SYSTEM TestSP
  (* Version 1.0, 2024-01-14, ADMIN *)
  APPLICATION TestSPApp
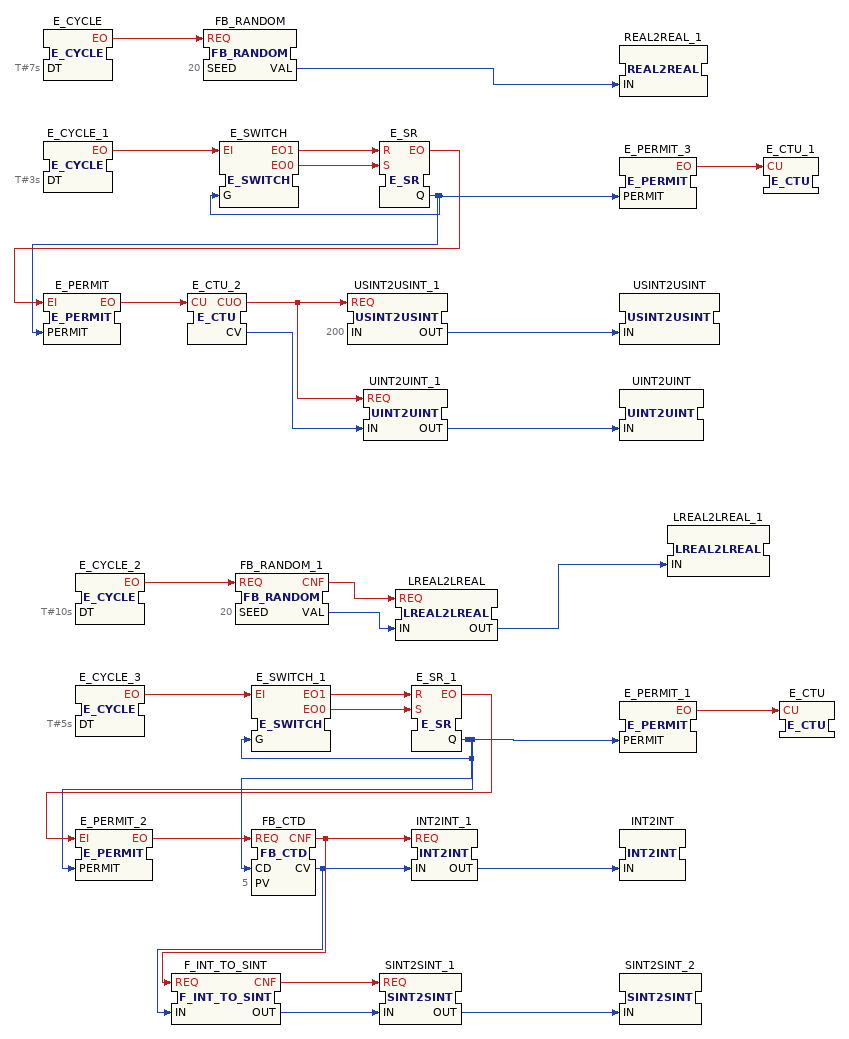
    FBS
      E_CYCLE : E_CYCLE(DT := T#7s);
      FB_RANDOM : FB_RANDOM(SEED := 20);
      E_CYCLE_1 : E_CYCLE(DT := T#3s);
      E_SWITCH : E_SWITCH;
      E_SR : E_SR;
      E_PERMIT : E_PERMIT;
      E_PERMIT_1 : E_PERMIT;
      E_CTU : E_CTU;
      E_CYCLE_2 : E_CYCLE(DT := T#10s);
      FB_RANDOM_1 : FB_RANDOM(SEED := 20);
      E_CYCLE_3 : E_CYCLE(DT := T#5s);
      E_SWITCH_1 : E_SWITCH;
      E_SR_1 : E_SR;
      E_PERMIT_2 : E_PERMIT;
      REAL2REAL_1 : REAL2REAL;
      E_PERMIT_3 : E_PERMIT;
      E_CTU_1 : E_CTU;
      UINT2UINT : UINT2UINT;
      INT2INT : INT2INT;
      SINT2SINT_1 : SINT2SINT;
      USINT2USINT : USINT2USINT;
      E_CTU_2 : E_CTU;
      UINT2UINT_1 : UINT2UINT;
      SINT2SINT_2 : SINT2SINT;
      INT2INT_1 : INT2INT;
      USINT2USINT_1 : USINT2USINT(IN := 200);
      LREAL2LREAL : LREAL2LREAL;
      LREAL2LREAL_1 : LREAL2LREAL;
      FB_CTD : FB_CTD(PV := 5);
      F_INT_TO_SINT : F_INT_TO_SINT;
    END_FBS
    EVENT_CONNECTIONS
      E_CYCLE.EO TO FB_RANDOM.REQ;
      E_SWITCH.EO1 TO E_SR.R;
      E_SWITCH.EO0 TO E_SR.S;
      E_SR.EO TO E_PERMIT.EI;
      E_CYCLE_1.EO TO E_SWITCH.EI;
      E_PERMIT_1.EO TO E_CTU.CU;
      E_PERMIT_3.EO TO E_CTU_1.CU;
      E_SR_1.EO TO E_PERMIT_2.EI;
      E_CYCLE_2.EO TO FB_RANDOM_1.REQ;
      E_SWITCH_1.EO1 TO E_SR_1.R;
      E_CYCLE_3.EO TO E_SWITCH_1.EI;
      E_SWITCH_1.EO0 TO E_SR_1.S;
      E_PERMIT.EO TO E_CTU_2.CU;
      E_CTU_2.CUO TO UINT2UINT_1.REQ;
      E_CTU_2.CUO TO USINT2USINT_1.REQ;
      FB_RANDOM_1.CNF TO LREAL2LREAL.REQ;
      E_PERMIT_2.EO TO FB_CTD.REQ;
      FB_CTD.CNF TO INT2INT_1.REQ;
      F_INT_TO_SINT.CNF TO SINT2SINT_1.REQ;
      FB_CTD.CNF TO F_INT_TO_SINT.REQ;
    END_CONNECTIONS
    DATA_CONNECTIONS
      E_SR.Q TO E_SWITCH.G;
      E_SR.Q TO E_PERMIT.PERMIT;
      E_SR_1.Q TO E_SWITCH_1.G;
      E_SR_1.Q TO E_PERMIT_2.PERMIT;
      E_SR.Q TO E_PERMIT_3.PERMIT;
      E_SR_1.Q TO E_PERMIT_1.PERMIT;
      FB_RANDOM.VAL TO REAL2REAL_1.IN;
      E_CTU_2.CV TO UINT2UINT_1.IN;
      INT2INT_1.OUT TO INT2INT.IN;
      SINT2SINT_1.OUT TO SINT2SINT_2.IN;
      USINT2USINT_1.OUT TO USINT2USINT.IN;
      UINT2UINT_1.OUT TO UINT2UINT.IN;
      FB_RANDOM_1.VAL TO LREAL2LREAL.IN;
      LREAL2LREAL.OUT TO LREAL2LREAL_1.IN;
      FB_CTD.CV TO INT2INT_1.IN;
      F_INT_TO_SINT.OUT TO SINT2SINT_1.IN;
      FB_CTD.CV TO F_INT_TO_SINT.IN;
      E_SR_1.Q TO FB_CTD.CD;
    END_CONNECTIONS
  END_APPLICATION
  DEVICE BeagleBoneBlack : BeagleBoneBlack(MGR_ID := "localhost:61500")
    {SET_ATTRIBUTE(Profile, HOLOBLOC)} (* device profile *)
    RESOURCE EMB_RES : EMB_RES
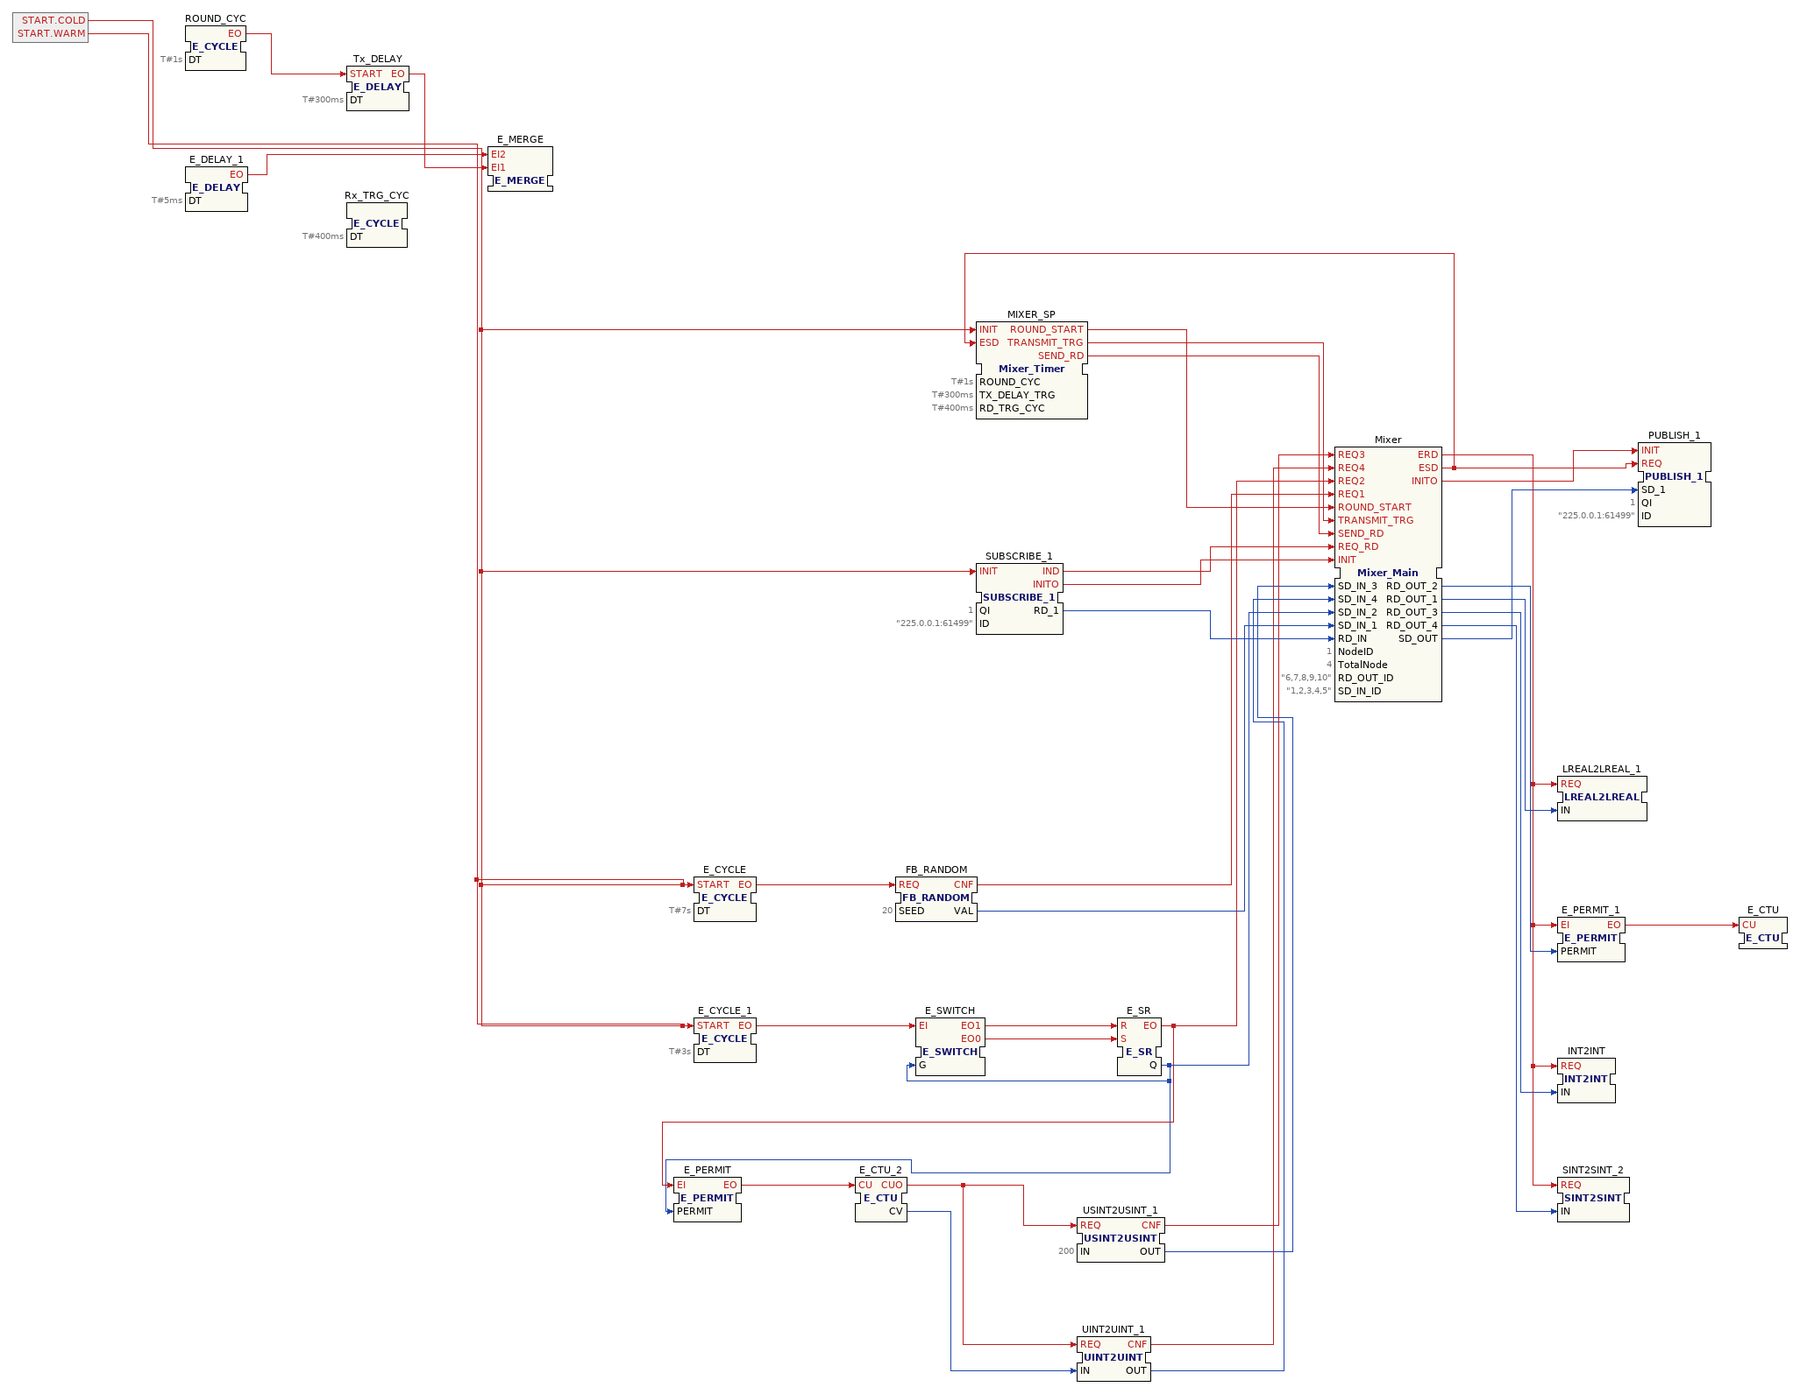
      FBS
        Mixer : Mixer_Main(NodeID := 1, TotalNode := 4, RD_OUT_ID := "6,7,8,9,10", SD_IN_ID := "1,2,3,4,5");
        Rx_TRG_CYC : E_CYCLE(DT := T#400ms);
        PUBLISH_1 : PUBLISH_1(QI := 1, ID := "225.0.0.1:61499");
        E_DELAY_1 : E_DELAY(DT := T#5ms);
        SUBSCRIBE_1 : SUBSCRIBE_1(QI := 1, ID := "225.0.0.1:61499");
        E_MERGE : E_MERGE;
        Tx_DELAY : E_DELAY(DT := T#300ms);
        ROUND_CYC : E_CYCLE(DT := T#1s);
        USINT2USINT_1 : USINT2USINT(IN := 200);
        UINT2UINT_1 : UINT2UINT;
        E_CTU_2 : E_CTU;
        E_CTU : E_CTU;
        E_PERMIT_1 : E_PERMIT;
        E_PERMIT : E_PERMIT;
        E_SR : E_SR;
        E_SWITCH : E_SWITCH;
        E_CYCLE_1 : E_CYCLE(DT := T#3s);
        FB_RANDOM : FB_RANDOM(SEED := 20);
        E_CYCLE : E_CYCLE(DT := T#7s);
        LREAL2LREAL_1 : LREAL2LREAL;
        INT2INT : INT2INT;
        SINT2SINT_2 : SINT2SINT;
        MIXER_SP : Mixer_Timer(ROUND_CYC := T#1s, TX_DELAY_TRG := T#300ms, RD_TRG_CYC := T#400ms);
      END_FBS
      EVENT_CONNECTIONS
        ROUND_CYC.EO TO Tx_DELAY.START;
        E_DELAY_1.EO TO E_MERGE.EI2;
        Tx_DELAY.EO TO E_MERGE.EI1;
        USINT2USINT_1.CNF TO Mixer.REQ3;
        UINT2UINT_1.CNF TO Mixer.REQ4;
        E_CTU_2.CUO TO UINT2UINT_1.REQ;
        E_CTU_2.CUO TO USINT2USINT_1.REQ;
        E_PERMIT_1.EO TO E_CTU.CU;
        Mixer.ERD TO E_PERMIT_1.EI;
        E_PERMIT.EO TO E_CTU_2.CU;
        E_SR.EO TO E_PERMIT.EI;
        E_SR.EO TO Mixer.REQ2;
        E_SWITCH.EO1 TO E_SR.R;
        E_SWITCH.EO0 TO E_SR.S;
        E_CYCLE_1.EO TO E_SWITCH.EI;
        START.COLD TO E_CYCLE_1.START;
        START.WARM TO E_CYCLE_1.START;
        FB_RANDOM.CNF TO Mixer.REQ1;
        E_CYCLE.EO TO FB_RANDOM.REQ;
        START.COLD TO E_CYCLE.START;
        START.WARM TO E_CYCLE.START;
        Mixer.ERD TO LREAL2LREAL_1.REQ;
        Mixer.ERD TO INT2INT.REQ;
        Mixer.ERD TO SINT2SINT_2.REQ;
        START.COLD TO MIXER_SP.INIT;
        Mixer.ESD TO MIXER_SP.ESD;
        MIXER_SP.ROUND_START TO Mixer.ROUND_START;
        MIXER_SP.TRANSMIT_TRG TO Mixer.TRANSMIT_TRG;
        MIXER_SP.SEND_RD TO Mixer.SEND_RD;
        SUBSCRIBE_1.IND TO Mixer.REQ_RD;
        Mixer.INITO TO PUBLISH_1.INIT;
        Mixer.ESD TO PUBLISH_1.REQ;
        SUBSCRIBE_1.INITO TO Mixer.INIT;
        START.COLD TO SUBSCRIBE_1.INIT;
      END_CONNECTIONS
      DATA_CONNECTIONS
        USINT2USINT_1.OUT TO Mixer.SD_IN_3;
        UINT2UINT_1.OUT TO Mixer.SD_IN_4;
        E_CTU_2.CV TO UINT2UINT_1.IN;
        E_SR.Q TO E_PERMIT.PERMIT;
        E_SR.Q TO Mixer.SD_IN_2;
        E_SR.Q TO E_SWITCH.G;
        FB_RANDOM.VAL TO Mixer.SD_IN_1;
        Mixer.RD_OUT_2 TO E_PERMIT_1.PERMIT;
        Mixer.RD_OUT_1 TO LREAL2LREAL_1.IN;
        Mixer.RD_OUT_3 TO INT2INT.IN;
        Mixer.RD_OUT_4 TO SINT2SINT_2.IN;
        SUBSCRIBE_1.RD_1 TO Mixer.RD_IN;
        Mixer.SD_OUT TO PUBLISH_1.SD_1;
      END_CONNECTIONS
    END_RESOURCE
  END_DEVICE
  DEVICE BeagleBoneBlack_1 : BeagleBoneBlack(MGR_ID := "localhost:61501")
    {SET_ATTRIBUTE(Profile, HOLOBLOC)} (* device profile *)
    RESOURCE EMB_RES : EMB_RES
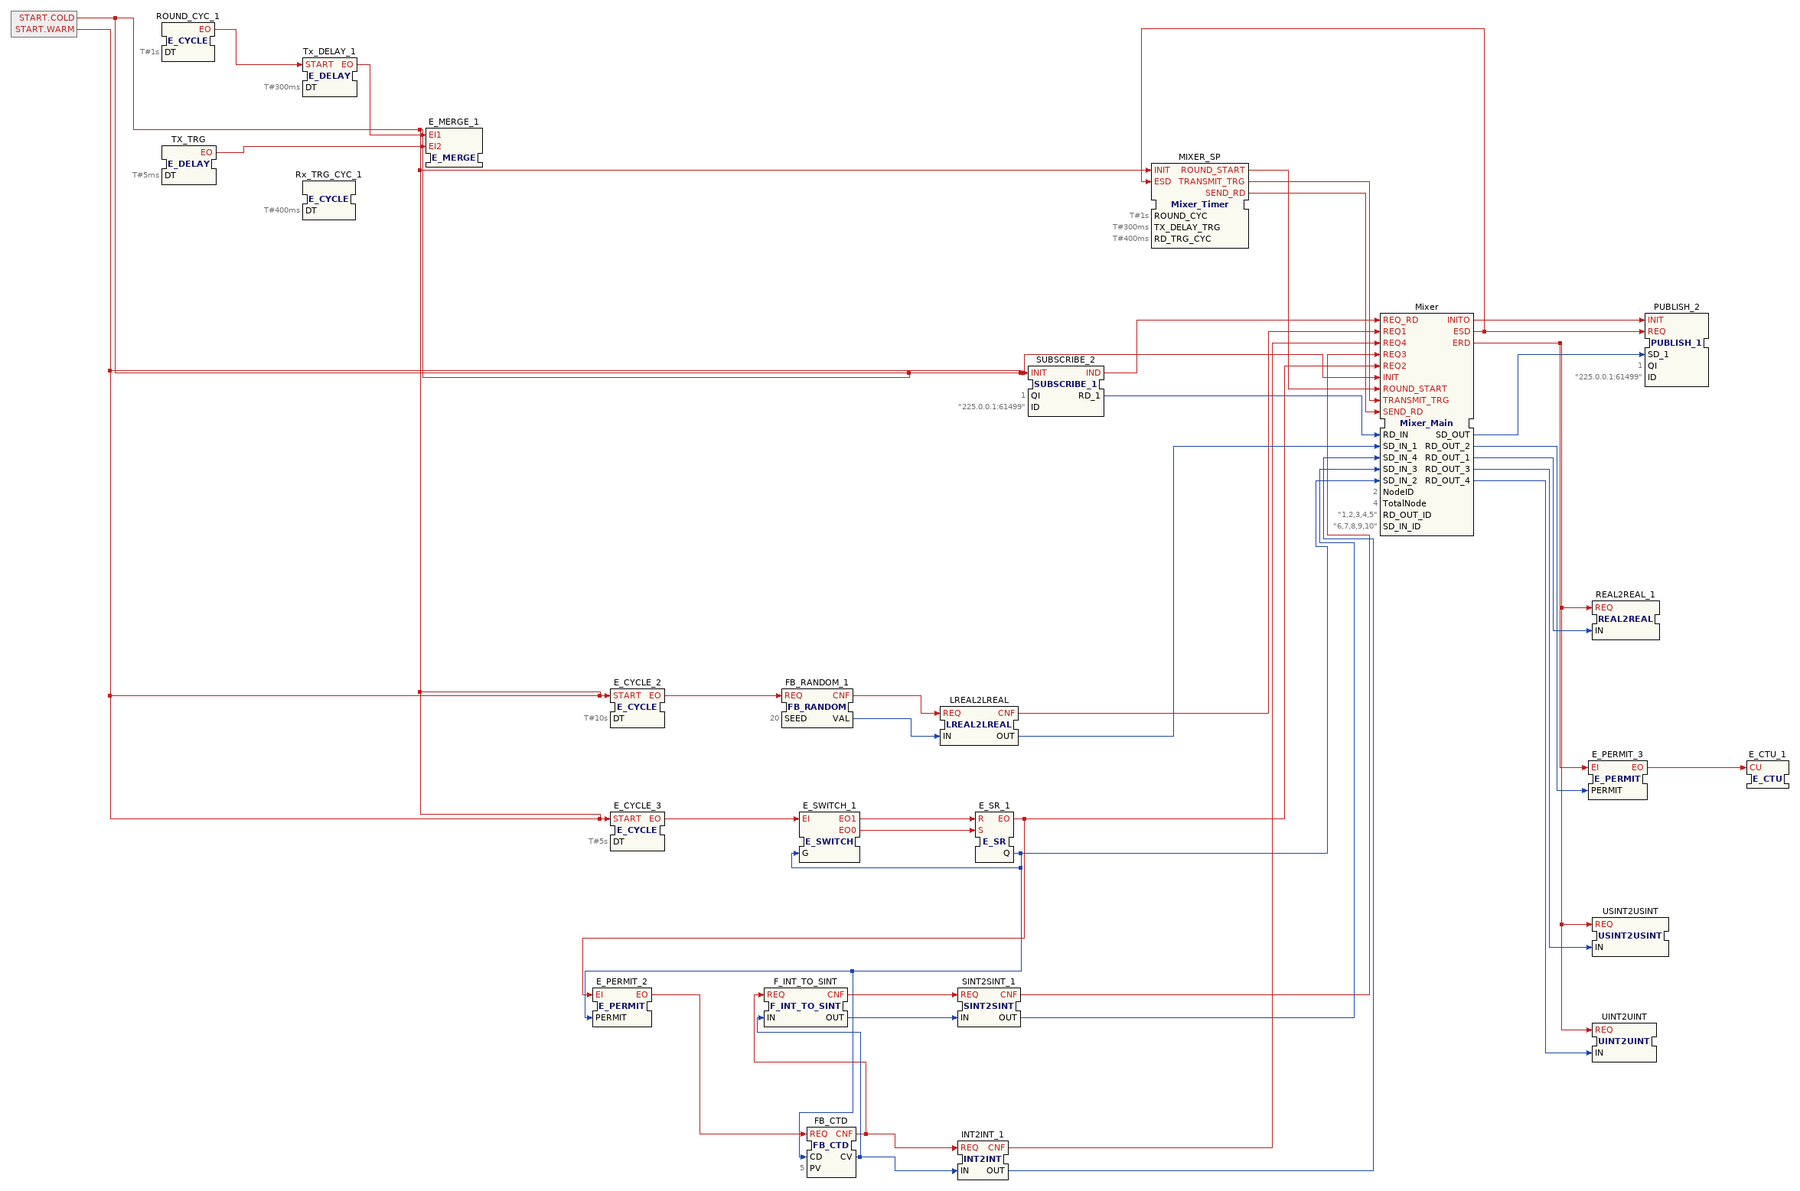
      FBS
        E_MERGE_1 : E_MERGE;
        Tx_DELAY_1 : E_DELAY(DT := T#300ms);
        TX_TRG : E_DELAY(DT := T#5ms);
        PUBLISH_2 : PUBLISH_1(QI := 1, ID := "225.0.0.1:61499");
        SUBSCRIBE_2 : SUBSCRIBE_1(QI := 1, ID := "225.0.0.1:61499");
        Mixer : Mixer_Main(NodeID := 2, TotalNode := 4, RD_OUT_ID := "1,2,3,4,5", SD_IN_ID := "6,7,8,9,10");
        Rx_TRG_CYC_1 : E_CYCLE(DT := T#400ms);
        ROUND_CYC_1 : E_CYCLE(DT := T#1s);
        F_INT_TO_SINT : F_INT_TO_SINT;
        FB_CTD : FB_CTD(PV := 5);
        LREAL2LREAL : LREAL2LREAL;
        INT2INT_1 : INT2INT;
        SINT2SINT_1 : SINT2SINT;
        E_CTU_1 : E_CTU;
        E_PERMIT_3 : E_PERMIT;
        E_PERMIT_2 : E_PERMIT;
        E_SR_1 : E_SR;
        E_SWITCH_1 : E_SWITCH;
        E_CYCLE_3 : E_CYCLE(DT := T#5s);
        FB_RANDOM_1 : FB_RANDOM(SEED := 20);
        E_CYCLE_2 : E_CYCLE(DT := T#10s);
        USINT2USINT : USINT2USINT;
        REAL2REAL_1 : REAL2REAL;
        UINT2UINT : UINT2UINT;
        MIXER_SP : Mixer_Timer(ROUND_CYC := T#1s, TX_DELAY_TRG := T#300ms, RD_TRG_CYC := T#400ms);
      END_FBS
      EVENT_CONNECTIONS
        Tx_DELAY_1.EO TO E_MERGE_1.EI1;
        ROUND_CYC_1.EO TO Tx_DELAY_1.START;
        Mixer.INITO TO PUBLISH_2.INIT;
        TX_TRG.EO TO E_MERGE_1.EI2;
        SUBSCRIBE_2.IND TO Mixer.REQ_RD;
        START.COLD TO SUBSCRIBE_2.INIT;
        START.WARM TO SUBSCRIBE_2.INIT;
        Mixer.ESD TO PUBLISH_2.REQ;
        FB_CTD.CNF TO F_INT_TO_SINT.REQ;
        LREAL2LREAL.CNF TO Mixer.REQ1;
        INT2INT_1.CNF TO Mixer.REQ4;
        FB_CTD.CNF TO INT2INT_1.REQ;
        SINT2SINT_1.CNF TO Mixer.REQ3;
        F_INT_TO_SINT.CNF TO SINT2SINT_1.REQ;
        E_PERMIT_3.EO TO E_CTU_1.CU;
        Mixer.ERD TO E_PERMIT_3.EI;
        E_PERMIT_2.EO TO FB_CTD.REQ;
        E_SR_1.EO TO Mixer.REQ2;
        E_SR_1.EO TO E_PERMIT_2.EI;
        E_SWITCH_1.EO1 TO E_SR_1.R;
        E_SWITCH_1.EO0 TO E_SR_1.S;
        E_CYCLE_3.EO TO E_SWITCH_1.EI;
        START.WARM TO E_CYCLE_3.START;
        START.COLD TO E_CYCLE_3.START;
        FB_RANDOM_1.CNF TO LREAL2LREAL.REQ;
        E_CYCLE_2.EO TO FB_RANDOM_1.REQ;
        START.WARM TO E_CYCLE_2.START;
        START.COLD TO E_CYCLE_2.START;
        Mixer.ERD TO REAL2REAL_1.REQ;
        Mixer.ERD TO UINT2UINT.REQ;
        Mixer.ERD TO USINT2USINT.REQ;
        START.COLD TO Mixer.INIT;
        START.COLD TO MIXER_SP.INIT;
        Mixer.ESD TO MIXER_SP.ESD;
        MIXER_SP.ROUND_START TO Mixer.ROUND_START;
        MIXER_SP.TRANSMIT_TRG TO Mixer.TRANSMIT_TRG;
        MIXER_SP.SEND_RD TO Mixer.SEND_RD;
      END_CONNECTIONS
      DATA_CONNECTIONS
        SUBSCRIBE_2.RD_1 TO Mixer.RD_IN;
        Mixer.SD_OUT TO PUBLISH_2.SD_1;
        FB_CTD.CV TO F_INT_TO_SINT.IN;
        LREAL2LREAL.OUT TO Mixer.SD_IN_1;
        INT2INT_1.OUT TO Mixer.SD_IN_4;
        FB_CTD.CV TO INT2INT_1.IN;
        SINT2SINT_1.OUT TO Mixer.SD_IN_3;
        F_INT_TO_SINT.OUT TO SINT2SINT_1.IN;
        E_SR_1.Q TO Mixer.SD_IN_2;
        E_SR_1.Q TO E_PERMIT_2.PERMIT;
        E_SR_1.Q TO FB_CTD.CD;
        E_SR_1.Q TO E_SWITCH_1.G;
        FB_RANDOM_1.VAL TO LREAL2LREAL.IN;
        Mixer.RD_OUT_2 TO E_PERMIT_3.PERMIT;
        Mixer.RD_OUT_1 TO REAL2REAL_1.IN;
        Mixer.RD_OUT_3 TO USINT2USINT.IN;
        Mixer.RD_OUT_4 TO UINT2UINT.IN;
      END_CONNECTIONS
    END_RESOURCE
  END_DEVICE
  MAPPINGS
    TestSPApp.F_INT_TO_SINT ON BeagleBoneBlack_1.EMB_RES.F_INT_TO_SINT;
    TestSPApp.FB_CTD ON BeagleBoneBlack_1.EMB_RES.FB_CTD;
    TestSPApp.LREAL2LREAL ON BeagleBoneBlack_1.EMB_RES.LREAL2LREAL;
    TestSPApp.USINT2USINT_1 ON BeagleBoneBlack.EMB_RES.USINT2USINT_1;
    TestSPApp.INT2INT_1 ON BeagleBoneBlack_1.EMB_RES.INT2INT_1;
    TestSPApp.UINT2UINT_1 ON BeagleBoneBlack.EMB_RES.UINT2UINT_1;
    TestSPApp.E_CTU_2 ON BeagleBoneBlack.EMB_RES.E_CTU_2;
    TestSPApp.SINT2SINT_1 ON BeagleBoneBlack_1.EMB_RES.SINT2SINT_1;
    TestSPApp.E_CTU_1 ON BeagleBoneBlack_1.EMB_RES.E_CTU_1;
    TestSPApp.E_PERMIT_3 ON BeagleBoneBlack_1.EMB_RES.E_PERMIT_3;
    TestSPApp.E_PERMIT_2 ON BeagleBoneBlack_1.EMB_RES.E_PERMIT_2;
    TestSPApp.E_SR_1 ON BeagleBoneBlack_1.EMB_RES.E_SR_1;
    TestSPApp.E_SWITCH_1 ON BeagleBoneBlack_1.EMB_RES.E_SWITCH_1;
    TestSPApp.E_CYCLE_3 ON BeagleBoneBlack_1.EMB_RES.E_CYCLE_3;
    TestSPApp.FB_RANDOM_1 ON BeagleBoneBlack_1.EMB_RES.FB_RANDOM_1;
    TestSPApp.E_CYCLE_2 ON BeagleBoneBlack_1.EMB_RES.E_CYCLE_2;
    TestSPApp.E_CTU ON BeagleBoneBlack.EMB_RES.E_CTU;
    TestSPApp.E_PERMIT_1 ON BeagleBoneBlack.EMB_RES.E_PERMIT_1;
    TestSPApp.E_PERMIT ON BeagleBoneBlack.EMB_RES.E_PERMIT;
    TestSPApp.E_SR ON BeagleBoneBlack.EMB_RES.E_SR;
    TestSPApp.E_SWITCH ON BeagleBoneBlack.EMB_RES.E_SWITCH;
    TestSPApp.E_CYCLE_1 ON BeagleBoneBlack.EMB_RES.E_CYCLE_1;
    TestSPApp.FB_RANDOM ON BeagleBoneBlack.EMB_RES.FB_RANDOM;
    TestSPApp.E_CYCLE ON BeagleBoneBlack.EMB_RES.E_CYCLE;
    TestSPApp.USINT2USINT ON BeagleBoneBlack_1.EMB_RES.USINT2USINT;
    TestSPApp.REAL2REAL_1 ON BeagleBoneBlack_1.EMB_RES.REAL2REAL_1;
    TestSPApp.UINT2UINT ON BeagleBoneBlack_1.EMB_RES.UINT2UINT;
    TestSPApp.LREAL2LREAL_1 ON BeagleBoneBlack.EMB_RES.LREAL2LREAL_1;
    TestSPApp.INT2INT ON BeagleBoneBlack.EMB_RES.INT2INT;
    TestSPApp.SINT2SINT_2 ON BeagleBoneBlack.EMB_RES.SINT2SINT_2;
  END_MAPPINGS
  SEGMENTS
    Ethernet : Ethernet;
  END_SEGMENTS
  LINKS
    BeagleBoneBlack => Ethernet;
    BeagleBoneBlack_1 => Ethernet;
  END_LINKS
END_SYSTEM
